INTERFACE ITF_Pomp

PROPERTY ActueelToerental : INT
GET
END_GET
SET
END_SET
END_PROPERTY

METHOD Open : BOOL
VAR_INPUT
END_VAR
END_METHOD

METHOD PompGoTo : INT
VAR_INPUT
	toerental : INT;
END_VAR
END_METHOD

PROPERTY StatePomp : E_PompState
GET
END_GET
SET
END_SET
END_PROPERTY

END_INTERFACE

(* stored: Version 1.1.0.1, ProductVersion 3.1.4026.8
   Itf ITF_Pomp: Id {9239626d-ca85-4ec3-a975-4f64db65a75e}
   Property ActueelToerental: Id {54c501b4-4fec-4cb7-abfd-20b8f37ebed2}
   Get Get: Id {cabaeb82-23e1-4a32-bf5f-6f61d552673b}
   Set Set: Id {85781121-3548-42f7-a59a-9b095738f2c6}
   Method Open: Id {296b4c6c-e3a0-49b2-9950-040b11a920d2}
   Method PompGoTo: Id {79f0a90a-1cff-424f-80fb-af47f655734a}
   Property StatePomp: Id {4a6177c8-326d-40bd-9103-d1160ee0e1b5}
   Get Get: Id {745e4efc-864f-4cd5-8b99-52464470cbad}
   Set Set: Id {bd88271f-02b4-40dc-b0b3-eee74b98a7c6} *)
